// TIA Portal project "VentiladorE3Siemens" (V14)

(* hardware
DEVICE "S7-1200 station_1"  S7-1200 Station
   slot 0: "Rack_0"  S7-1200 Rack  Rack  V1.0
   slot 1: "PLC_1"  CPU 1214C DC/DC/DC  6ES7 214-1AG40-0XB0  V4.2
*)

// ===== PLC "PLC_1"  CPU 1214C DC/DC/DC =====

VAR_GLOBAL   // PLC tag table "Default tag table"
   "Liga" AT %I0.1 : Bool;
   "Desliga" AT %I0.2 : Bool;
   "Desliga E3" AT %M0.1 : Bool;
   "Ventilador" AT %Q1.0 : Bool;
   "Liga E3" AT %M0.2 : Bool;
   "Vent" AT %Q0.0 : Bool;
   "Tag_1" AT %M0.3 : Bool;
END_VAR

ORGANIZATION_BLOCK "Main"   // OB1, LAD, ProgramCycle
TITLE = "Main Program Sweep (Cycle)"
{ S7_Optimized_Access := 'TRUE' }
VERSION : 0.1
   VAR_INPUT
      Initial_Call : Bool;   // Initial call of this OB
      Remanence : Bool;   // =True, if remanent data are available
   END_VAR
BEGIN

REGION Network 1
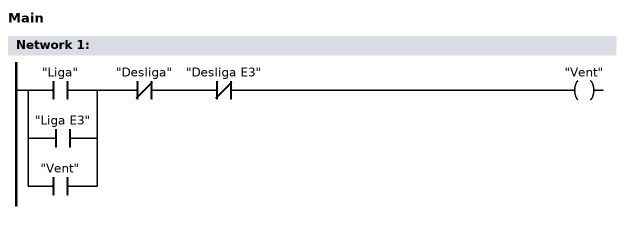
   RUNG wire#powerrail
      Contact( "Liga" )
      wire#w1
      I_Contact( "Desliga" )
      I_Contact( "Desliga E3" )
      Coil( "Vent" )
   END_RUNG
   RUNG wire#powerrail
      Contact( "Liga E3" )
   END_RUNG wire#w1
   RUNG wire#powerrail
      Contact( "Vent" )
   END_RUNG wire#w1
   // the same network as SCL:
   "Vent" := ("Liga" OR "Liga E3" OR "Vent") AND NOT "Desliga" AND NOT "Desliga E3";
END_REGION
END_ORGANIZATION_BLOCK